// TIA Portal V17 export
// export: Created 2022-02-03T14:45:16.0334072Z, ExportSetting WithDefaults, DisplayName Totally Integrated Automation Portal, DisplayVersion V17, DisplayName TIA Portal Openness, DisplayVersion V17, DisplayName TIA Portal Version Control Interface, DisplayVersion V17, DisplayName SINAMICS Startdrive Advanced, DisplayVersion V17, DisplayName SINAMICS Startdrive G130, G150, S120, S150, SINAMICS MV, S210, DisplayVersion V17, DisplayName SINAMICS Startdrive G110M, G120, G120C, G120D, G120P, G115D, DisplayVersion V17, DisplayName STEP 7 Professional, DisplayVersion V17, DisplayName STEP 7 Safety, DisplayVersion V17, DisplayName WinCC Advanced, DisplayVersion V17
DATA_BLOCK "ConveyorData"   // DB2
VERSION : 0.1
// stored: Access Published, AutoNumber true, DBAccessibleFromOPCUA true, DBAccessibleFromWebserver true, IsOnlyStoredInLoadMemory false, IsRetainMemResEnabled false, IsWriteProtectedInAS false, MemoryReserve 100
   VAR
      occupiedBay : Array["FIRSTBAY".."LASTBAY"] of Bool;
      weightSimulation : UInt;
      weightOk : Bool;
      instIECTimer : IEC_TIMER;
      getError { S7_SetPoint := 'True'} : ErrorStruct;
   END_VAR
BEGIN
END_DATA_BLOCK
